// TIA Portal project "Height Sorting" (V16)

(* hardware
DEVICE "S7300/ET200M station_1"  S7-300 station
   slot 0: "Rail_0"  Rail  6ES7 390-1***0-0AA0
   slot 2: "PLC_1"  CPU 312  6ES7 312-1AE13-0AB0  V2.6
      slot 0: "MPI interface_1"  X1
*)

// ===== PLC "PLC_1"  CPU 312 =====

VAR_GLOBAL   // PLC tag table "Default tag table"
   "start" AT %I0.0 : Bool;
   "stop" AT %I0.1 : Bool;
   "sensor1" AT %I0.2 : Bool;
   "sensor2" AT %I0.3 : Bool;
   "front" AT %I0.4 : Bool;
   "Conv - 1" AT %Q0.0 : Bool;
   "pusher" AT %Q0.1 : Bool;
   "M0" AT %M0.0 : Bool;
   "M1" AT %M0.1 : Bool;
   "T1" AT %M0.2 : Bool;
   "T2" AT %M0.3 : Bool;
   "Conv - 2" AT %Q0.2 : Bool;
END_VAR

ORGANIZATION_BLOCK "Main"   // OB1, LAD
TITLE = "Main Program Sweep (Cycle)"
{ S7_Optimized_Access := 'FALSE' }
VERSION : 0.1
   VAR_TEMP
      OB1_EV_CLASS : Byte;   // Bits 0-3 = 1 (Coming event), Bits 4-7 = 1 (Event class 1)
      OB1_SCAN_1 : Byte;   // 1 (Cold restart scan 1 of OB 1), 3 (Scan 2-n of OB 1)
      OB1_PRIORITY : Byte;   // Priority of OB Execution
      OB1_OB_NUMBR : Byte;   // 1 (Organization block 1, OB1)
      OB1_RESERVED_1 : Byte;   // Reserved for system
      OB1_RESERVED_2 : Byte;   // Reserved for system
      OB1_PREV_CYCLE : Int;   // Cycle time of previous OB1 scan (milliseconds)
      OB1_MIN_CYCLE : Int;   // Minimum cycle time of OB1 (milliseconds)
      OB1_MAX_CYCLE : Int;   // Maximum cycle time of OB1 (milliseconds)
      OB1_DATE_TIME : Date_And_Time;   // Date and time OB1 started
   END_VAR
   VAR_TEMP   // added for the SCL form of the ladder/FBD networks
      _w1 : Bool;
      _w2 : Bool;
   END_VAR
BEGIN

REGION Network 1: Start and stop
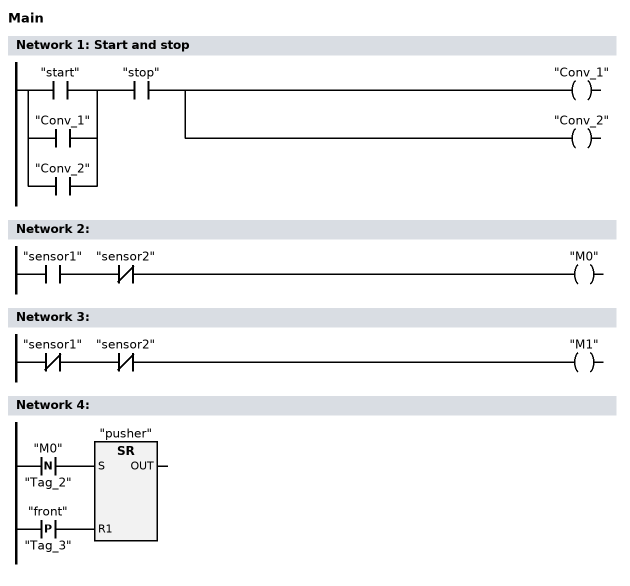
   RUNG wire#powerrail
      Contact( "start" )
      wire#w1
      Contact( "stop" )
      wire#w2
      Coil( "Conv_1" )
   END_RUNG
   RUNG wire#powerrail
      Contact( "Conv_1" )
   END_RUNG wire#w1
   RUNG wire#powerrail
      Contact( "Conv_2" )
   END_RUNG wire#w1
   RUNG wire#w2
      Coil( "Conv_2" )
   END_RUNG
   // the same network as SCL:
   "Conv_1" := ("start" OR "Conv_1" OR "Conv_2") AND "stop";
   "Conv_2" := "Conv_1";
END_REGION

REGION Network 2
   RUNG wire#powerrail
      Contact( "sensor1" )
      I_Contact( "sensor2" )
      Coil( "M0" )
   END_RUNG
   // the same network as SCL:
   "M0" := "sensor1" AND NOT "sensor2";
END_REGION

REGION Network 3
   RUNG wire#powerrail
      I_Contact( "sensor1" )
      I_Contact( "sensor2" )
      Coil( "M1" )
   END_RUNG
   // the same network as SCL:
   "M1" := NOT "sensor1" AND NOT "sensor2";
END_REGION

REGION Network 4
   RUNG wire#powerrail
      N_Contact(operand := "M0", bit := "Tag_2")
      S_SR(operand := "pusher", r1 := wire#w1)
   END_RUNG
   RUNG wire#powerrail
      P_Contact(operand := "front", bit := "Tag_3")
   END_RUNG wire#w1
   // the same network as SCL:
   #_w1 := NOT "M0" AND "Tag_2";   // falling edge of "M0"
   "Tag_2" := "M0";
   #_w2 := "front" AND NOT "Tag_3";   // rising edge of "front"
   "Tag_3" := "front";
   IF #_w1 THEN
       "pusher" := TRUE;   // SR flip-flop
   END_IF;
   IF #_w2 THEN "pusher" := FALSE; END_IF;
END_REGION
END_ORGANIZATION_BLOCK